(* IEC 61131-3 sources: inproshop/Team-Test6_exported/OP50/1.Global, 7 files *)

(* ---- DB5000_Control.st ---- *)
VAR_GLOBAL
	Mode:Str_Mode;
	HMI:Str_HMI;
END_VAR
VAR_GLOBAL RETAIN PERSISTENT
	Machine   : Str_Machine;
END_VAR

(* ---- DB5002_Recipe.st ---- *)
VAR_GLOBAL
END_VAR
VAR_GLOBAL RETAIN PERSISTENT

	RecipeChangePmt   : BOOL;	//配方允许切换
	ParameterChangePmt   : BOOL;	//参数允许更改
	RecipeNumTemp  : INT;	//HMI选中还未保存到PLC的编号.
	RecipeNum   : INT;	//配方元素编号.
	RecipeName   : STRING(20);	//配方元素名称.
	RecipeNameTemp   : STRING(20);	//HMI头部显示当前配方名称
	RecipeOk  : BOOL;//配方可用
	DownLoad   : BOOL;//配方下载
	TypeDataCur  : Str_OP30_Recipe;//当前配方
	TypeData   : ARRAY [0..20] OF Str_OP30_Recipe;//配方数据
END_VAR

(* ---- DB5003_Count.st ---- *)
VAR_GLOBAL RETAIN PERSISTENT
	Total  : Str_Count;//总计数
	OK  : Str_Count;//OK计数
	NG   : Str_Count;//NG计数
END_VAR
VAR_GLOBAL
	Yield : REAL;//良品率
	Clear : BOOL;//清除计数
END_VAR

(* ---- DB5005_Communication.st ---- *)
VAR_GLOBAL
	TcpClient:ARRAY[0..9] OF Str_TcpClient;
	TcpSever:ARRAY[0..9] OF Str_TcpClient;
	From_OPXX    :Str_OP80_TO_OPXX;
	TO_OPXX    :Str_OPXX_TO_OP80;
	FromMaster  :Str_FromMaster;
END_VAR

(* ---- DB5050_DriveControl.st ---- *)
VAR_GLOBAL RETAIN PERSISTENT
	CylCtrl   : ARRAY [0..63] OF Str_Cylinder;
	VacCtrl   : ARRAY [0..32] OF Str_Cylinder;
	AxisCtrl  : ARRAY [0..16] OF Str_Axis;
	Sensor  : ARRAY [0..32] OF Str_Sensor;
	CamCtrl  : ARRAY [1..3] OF Str_CamControl;
END_VAR

VAR_GLOBAL
	DoubleStart:ARRAY [1..4] OF Str_DoubleStart;
	Epson : ARRAY [1..10] OF Str_Epson;
	Kuka : ARRAY [1..2] OF Str_Kuka6;
	Rotdisk:ARRAY [1..1] OF Str_Rotdisk;
	Stopper:ARRAY [1..20] OF Str_Stopper;
	Motor:ARRAY [1..10] OF Str_Motor;
	AI:ARRAY [0..20] OF Str_AI;
	AAS:ARRAY [1..1] OF Str_AAS;
	HeatCtrl : ARRAY [1..1] OF Str_Heating;
	PalletCtrl : ARRAY [0..3] OF Str_Palletizing;
END_VAR

(* ---- DB5070_Fault.st ---- *)
VAR_GLOBAL
	Estop:Str_OP30_FaultEstop;//紧急停止类报警
	Stop:Str_OP30_Faultstop;//暂停类报警
	Run:Str_OP30_FaultRun;//警告类报警
	EstopTotal:BOOL;//急停报警汇总
	StopTotal:BOOL;//暂停报警汇总
	RunTotal:BOOL;//警告汇总
END_VAR

(* ---- DB5090_Other.st ---- *)
VAR_GLOBAL RETAIN PERSISTENT
	{attribute 'ElemComment':='(),(上料机械臂取料夹爪),(上料机械臂放料夹爪),(缓存台1),(缓存台2),(缓存台3),(缓存台4),(测试台1),(测试台2),(测试台3),(测试台4),(下料机械臂),4()'}
	StationData   : ARRAY [0..15] OF Str_OP30_StationData;
END_VAR
